TYPE ST_AccessConnectionInfo :
STRUCT
	Path:STRING(255);
END_STRUCT
END_TYPE

(* stored: Version 1.1.0.1, ProductVersion 3.1.4024.2
   DUT ST_AccessConnectionInfo: Id {e2d40b3d-09f9-4468-bf04-606c05ed5dc9} *)
